
FUNCTION CB_gt_date : BOOL


TITLE = ' Test Whether IN0 is strictly greater than IN1 '
VERSION : '1.0'
AUTHOR  : CB
NAME    : gt_date
FAMILY  : TNI

VAR_INPUT
    IN0 : DATE;
    IN1 : DATE;
END_VAR

BEGIN

CB_gt_date := (IN0 > IN1);

END_FUNCTION
